// Mitsubishi GX Works2 project: PLC_theoretic_B   PLC: FX3G

// global labels: Global1
VAR_GLOBAL
  choose_big AT X001 : BOOL;
  light_choose_big AT Y001 : BOOL;
  choose_mid AT X002 : BOOL;
  choose_small AT X003 : BOOL;
  light_choose_mid AT Y002 : BOOL;
  light_choose_small AT Y003 : BOOL;
  big_timer AT TC250 : BOOL;
END_VAR
VAR_GLOBAL CONSTANT
  big_time : INT := K150;
  mid_time : INT := K100;
END_VAR
VAR_GLOBAL
  mid_timer AT TC252 : BOOL;
  small_timer AT TC254 : BOOL;
END_VAR
VAR_GLOBAL CONSTANT
  small_time : INT := K50;
END_VAR
VAR_GLOBAL
  mid_timer_end AT TS252 : BOOL;
  small_timer_end AT TS250 : BOOL;
  big_timer_end AT TS254 : BOOL;
  drinks_filled_counter AT CC1 : BOOL;
END_VAR
VAR_GLOBAL CONSTANT
  target_drinks_filled : INT := 3;
END_VAR
VAR_GLOBAL
  above_10 AT X004 : BOOL;
  above_20 AT X005 : BOOL;
  end_of_fill AT Y004 : BOOL;
  drink_filled AT CN1 : INT;
  drinks_fill_finish AT CS1 : BOOL;
  start_day AT X007 : BOOL;
  day_started AT Y007 : BOOL;
END_VAR

// task Task_01 (event TRUE, interval 0, priority 31): POU_01

PROGRAM POU_01
(* structured ladder/FBD written out as ST: instructions are called as NAME(EN, inputs, outputs); _pN, _eN, _tN stand for wires *)
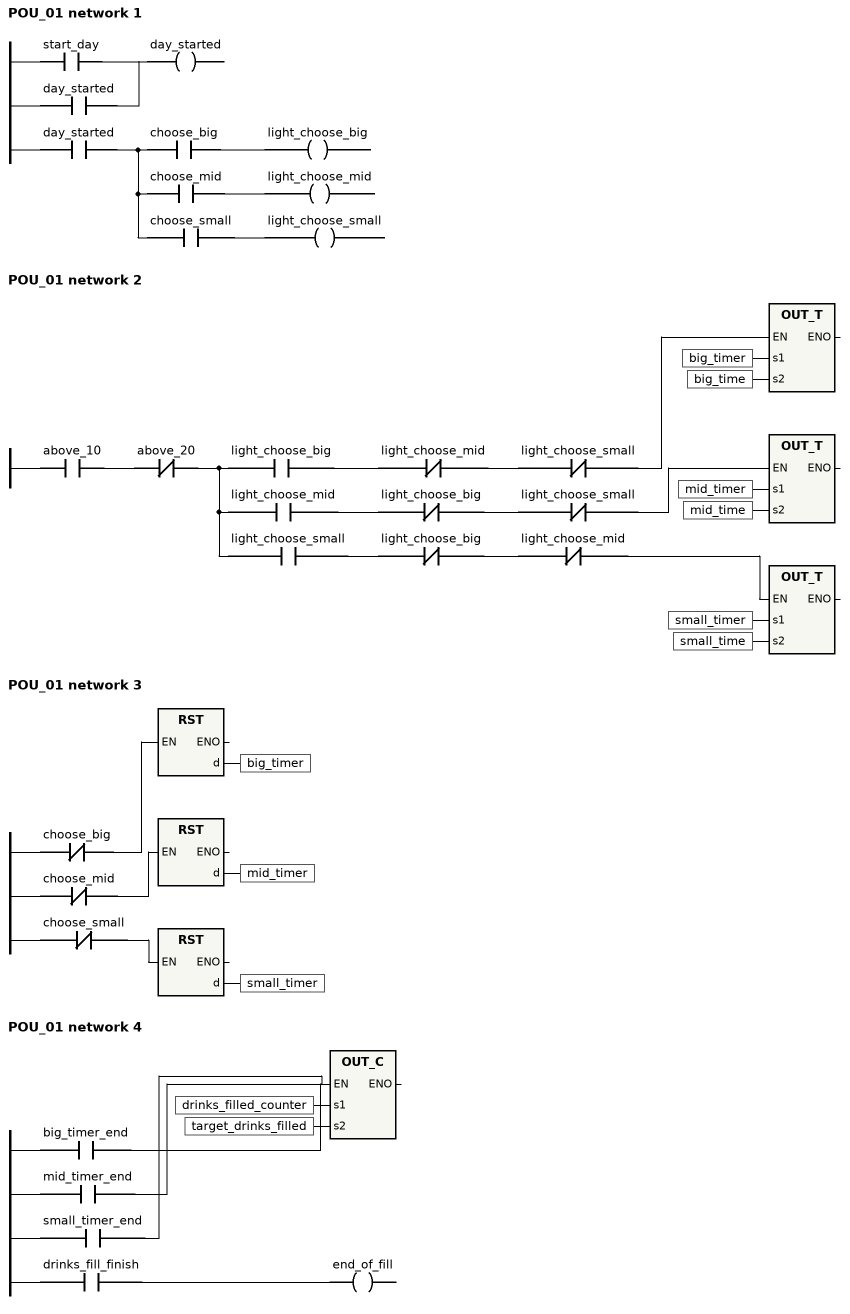
(* network 1 *)
day_started := start_day OR day_started;
light_choose_big := day_started AND choose_big;
light_choose_mid := day_started AND choose_mid;
light_choose_small := day_started AND choose_small;
(* network 2 *)
_p1 := above_10 AND NOT above_20;
OUT_T(_p1 AND light_choose_big AND NOT light_choose_mid AND NOT light_choose_small, big_timer, big_time);
OUT_T(_p1 AND light_choose_mid AND NOT light_choose_big AND NOT light_choose_small, mid_timer, mid_time);
OUT_T(_p1 AND light_choose_small AND NOT light_choose_big AND NOT light_choose_mid, small_timer, small_time);
(* network 3 *)
RST(NOT choose_big, big_timer);
RST(NOT choose_mid, mid_timer);
RST(NOT choose_small, small_timer);
(* network 4 *)
OUT_C(big_timer_end OR mid_timer_end OR small_timer_end, drinks_filled_counter, target_drinks_filled);
end_of_fill := drinks_fill_finish;
END_PROGRAM
